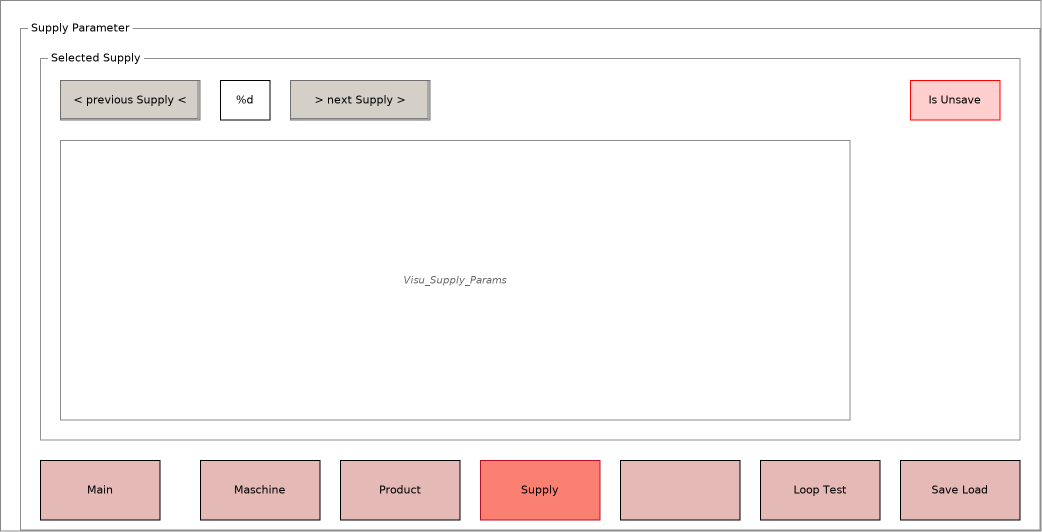
VISUALIZATION Visu_Supply  // 1042x532
    GroupBox (20,20 1020x510), "Supply Parameter"
        Rectangle (20,440 120x60), "Main"
            OnMouseClick: change screen: Visu_Main
        Rectangle (880,440 120x60), "Save Load"
            OnMouseClick: change screen: Visu_SaveLoad
        Rectangle (320,440 120x60), "Product"
            OnMouseClick: change screen: Visu_PParam
        Rectangle (180,440 120x60), "Maschine"
            OnMouseClick: change screen: Visu_MParam
        Rectangle (460,440 120x60), "Supply"
            OnMouseClick: change screen: Visu_Supply
        Rectangle (600,440 120x60)
        Rectangle (740,440 120x60), "Loop Test"
            OnMouseClick: change screen: Visu_LoopTest
        GroupBox (20,30 980x390), "Selected Supply"
            Rectangle (180,30 50x40), "%d", text variable: nSupplyCnt
            Button (20,30 140x40), "< previous Supply <"
                OnMouseClick: execute { nSupplyCnt:= MAX(cnPfwAppSupplyFirst, nSupplyCnt-1); }
            Button (250,30 140x40), "> next Supply >"
                OnMouseClick: execute { nSupplyCnt:= MIN(cnPfwAppSupplyLast, nSupplyCnt+1); }
            Rectangle (870,30 90x40), "Is Unsave", invisible if: Not stParamsUnsave.supply[nSupplyCnt]
                OnMouseClick: execute { stPfwSupplyLineCfg[nSupplyCnt].SaveDelay:=1000; stParamsUnsave.supply[nSupplyCnt]:=FALSE; }
            Frame (20,90 790x280)
                shows Visu_Supply_Params()
                shows Visu_MParam_ENUM()
                shows Visu_MParam_BOOL()
                shows Visu_MParam_INT()
END_VISUALIZATION

(* stored: Version 1.1.0.1, ProductVersion 3.1.4024.12
   Visu Visu_Supply: Id {4fdfc5f9-64e5-49b3-a601-19969aed2846} *)
